Staubli VAL3: ALGORITH.pjx

--- ALGORITH.pjx ---
Parameters version=s7.3.1 stackSize=5000 millimeterUnit=true
Program file=ArcLength.pgx
Program file=Axis1Offset.pgx
Program file=ChangeCirPoint.pgx
Program file=ChangeCpoint.pgx
Program file=ChangeLength.pgx
Program file=CirClePoint.pgx
Program file=Circumcircle.pgx
Program file=Cshape.pgx
Program file=CutIn.pgx
Program file=CutOut.pgx
Program file=EllipsePoint.pgx
Program file=Facula.pgx
Program file=GetArcAngle.pgx
Program file=GetArcLength.pgx
Program file=GetClockwise.pgx
Program file=GetCutLength.pgx
Program file=GetWeldId.pgx
Program file=GetWeldReturn.pgx
Program file=HexagonPoint.pgx
Program file=Inscribedcircle.pgx
Program file=LineSym.pgx
Program file=LineSymArray.pgx
Program file=NoCloseShape.pgx
Program file=PentaclePoint.pgx
Program file=PentagonPoint.pgx
Program file=ReadMe.pgx
Program file=RectanglePoint.pgx
Program file=RegulPoint.pgx
Program file=SetFrame.pgx
Program file=start.pgx
Program file=stop.pgx
Program file=TrianglePoint.pgx
Program file=TubePoint.pgx
Data file=Algorith.dtx

--- ALGORITH.dtx ---
trsf trCut[100]
num nThickRadio = 100

--- start.pgx ---
program start()
  local trsf l_trTrsf[3]
  local trsf l_trTrsf1
  local num l_nNum
  local bool l_bBool
begin
  l_trTrsf[0]={0,1,0,0,0,0}
   l_trTrsf[1]={0,0,1,0,0,0}
   l_trTrsf[2]={1,0,0,0,0,0}



  call Circumcircle(l_trTrsf,l_trTrsf1,l_nNum,l_bBool)
  if !l_bBool
    popUpMsg("")
  else
    popUpMsg(toString(".5",l_nNum))
  endIf




end

--- ArcLength.pgx ---
public program ArcLength(trsf x_trFirst, trsf x_trCenter, trsf x_trEnd, num& x_nLength)
  local trsf l_trTrsf[3]
  local bool l_bBool
begin


  //获得圆弧长度
  //如果报错,那么就返回值为0


  x_nLength=0

  l_trTrsf[0]=x_trFirst
  l_trTrsf[1]=x_trCenter
  l_trTrsf[2]=x_trEnd

  call GetArcLength(l_trTrsf,x_nLength,l_bBool)
  if !l_bBool
    x_nLength=0
  endIf



end

--- Axis1Offset.pgx ---
public program Axis1Offset(pointRx& x_pP[], num x_nOffset, tool x_tTool)
  local num l_nNum
  local bool l_bMC
  local num l_nValue[3]
  local joint l_jJ
  local point l_pPoint
  local frame l_fFrame
begin
  if size(x_pP)<3
    return
  endIf

  for l_nNum=10 to size(x_pP)-3
    l_nValue[0]=(x_pP[l_nNum].trsf.x-x_pP[l_nNum+1].trsf.x)/(x_pP[l_nNum].trsf.x-x_pP[l_nNum+2].trsf.x)
    l_nValue[1]=(x_pP[l_nNum].trsf.y-x_pP[l_nNum+1].trsf.y)/(x_pP[l_nNum].trsf.y-x_pP[l_nNum+2].trsf.y)
    l_nValue[2]=(x_pP[l_nNum].trsf.z-x_pP[l_nNum+1].trsf.z)/(x_pP[l_nNum].trsf.z-x_pP[l_nNum+2].trsf.z)

    if l_nValue[0]!=l_nValue[1] or l_nValue[0]!=l_nValue[2]

      if !pointToJoint(x_tTool,herej(),x_pP[l_nNum],l_jJ)
        popUpMsg("转换出错")
        disablePower()
        return
      else
        l_jJ.j1=l_jJ.j1+x_nOffset
        link(l_fFrame,world)
        link(l_pPoint,world)
        l_pPoint.trsf=position(x_pP[l_nNum],world)

        l_fFrame.trsf=l_pPoint.trsf*!x_pP[l_nNum].trsf
        l_pPoint=jointToPoint(x_tTool,l_fFrame,l_jJ)
        x_pP[l_nNum].trsf=l_pPoint.trsf
      endIf




    endIf




  endFor

















end

--- ChangeCirPoint.pgx ---
public program ChangeCirPoint(trsf x_trCenter, num x_nDia, trsf& x_trSource, trsf x_trSupport, bool& x_bRes)
  local frame l_fFrame
  local point l_pPoint[3]
begin
  //根据边长和圆心点来修改相应的点。

  x_bRes=false

  if x_nDia<=0
    return
  endIf

  l_pPoint[0].trsf=x_trCenter
  l_pPoint[1].trsf=x_trSource
  l_pPoint[2].trsf=x_trSupport

  link(l_pPoint[0],world)
  link(l_pPoint[1],world)
  link(l_pPoint[2],world)
  link(l_fFrame,world)

  if setFrame(l_pPoint[0],l_pPoint[1],l_pPoint[2],l_fFrame)!=0
    return
  endIf

  l_pPoint[1].trsf=position(l_pPoint[1],l_fFrame)
  l_pPoint[1].trsf.x=x_nDia/2
  link(l_pPoint[1],l_fFrame)
  x_trSource=position(l_pPoint[1],world)
  x_bRes=true

end

--- ChangeCpoint.pgx ---
public program ChangeCpoint(trsf& x_trSource[], num x_nDia, bool& x_bRes)
  local trsf l_trTrsf
  local num l_nDia
  local num l_nNum
begin
  //根据直径来修改点的数值
  //外接圆

  //先根据三点来获得圆心点，然后根据三个点来求的圆心与三个点的长度。



  x_bRes=false

  if size(x_trSource)!=3
    return
  endIf


  call Circumcircle(x_trSource,l_trTrsf,l_nDia,x_bRes)
  if !x_bRes
    return
  endIf

  for l_nNum=0 to 2
    call ChangeCirPoint(l_trTrsf,x_nDia,x_trSource[l_nNum],x_trSource[sel(l_nNum==2,0,l_nNum+1)],x_bRes)
    if !x_bRes
      return
    endIf
  endFor

end

--- ChangeLength.pgx ---
public program ChangeLength(pointRx& x_trSource[], num& x_nLength[])
  local num l_nBuff[2]
begin


  //参数合法化处理
  if size(x_trSource)<3
    return
  endIf

  l_nBuff[0]=distance(x_trSource[0].trsf,x_trSource[1].trsf)
  l_nBuff[1]=distance(x_trSource[2].trsf,x_trSource[1].trsf)


  if x_nLength[1]<=0 or x_nLength[0]<=0 or l_nBuff[0]<=0 or l_nBuff[1]<=0
    return
  endIf



  x_trSource[0].trsf.x=(x_trSource[0].trsf.x-x_trSource[1].trsf.x)/l_nBuff[0]*x_nLength[0]+x_trSource[1].trsf.x
  x_trSource[0].trsf.y=(x_trSource[0].trsf.y-x_trSource[1].trsf.y)/l_nBuff[0]*x_nLength[0]+x_trSource[1].trsf.y
  x_trSource[0].trsf.z=(x_trSource[0].trsf.z-x_trSource[1].trsf.z)/l_nBuff[0]*x_nLength[0]+x_trSource[1].trsf.z

  x_trSource[2].trsf.x=(x_trSource[2].trsf.x-x_trSource[1].trsf.x)/l_nBuff[1]*x_nLength[1]+x_trSource[1].trsf.x
  x_trSource[2].trsf.y=(x_trSource[2].trsf.y-x_trSource[1].trsf.y)/l_nBuff[1]*x_nLength[1]+x_trSource[1].trsf.y
  x_trSource[2].trsf.z=(x_trSource[2].trsf.z-x_trSource[1].trsf.z)/l_nBuff[1]*x_nLength[1]+x_trSource[1].trsf.z









end

--- CirClePoint.pgx ---
public program CirClePoint(trsf x_trCenter, num x_nDia, trsf& x_trDest[], bool& x_bRes)
  local num l_nNum
  local frame l_fFrame
  local point l_pP
begin
  //由圆心直径获得圆的四个点
  //是通过逆时针来获得

  x_bRes=false

  if x_nDia<=0
    return
  endIf

  link(l_fFrame,world)
  l_fFrame.trsf=x_trCenter
  link(l_pP,l_fFrame)


  //第一个点
  l_pP.trsf={0,0,0,0,0,0}
  l_pP.trsf.y=-x_nDia/2
  x_trDest[0]=position(l_pP,world)


  //第二个点
  l_pP.trsf={0,0,0,0,0,0}
  l_pP.trsf.x=x_nDia/2
  x_trDest[1]=position(l_pP,world)



  //第三个点
  l_pP.trsf={0,0,0,0,0,0}
  l_pP.trsf.y=x_nDia/2
  x_trDest[2]=position(l_pP,world)


  //第四个点
  l_pP.trsf={0,0,0,0,0,0}
  l_pP.trsf.x=-x_nDia/2
  x_trDest[3]=position(l_pP,world)

   x_trDest[4]= x_trDest[0]





  //圆心点
  x_trDest[20]=x_trCenter

  x_bRes=true

  //辅助点
  l_pP.trsf={0,0,0,0,0,0}
  l_pP.trsf.y=-x_nDia/2
    l_pP.trsf.x=x_nDia/2
  x_trDest[9]=position(l_pP,world)






end

--- Circumcircle.pgx ---
public program Circumcircle(trsf& x_trSource[], trsf& x_trCenter, num& x_nDia, bool& x_bRes)
  local point l_pPoint[3]
  local num l_ni
  local frame l_fFrame
  local point l_pCenter
  local num x1
  local num x2
  local num x3
  local num y1
  local num y2
  local num y3
begin
  //由圆的三点获得圆的圆心与直径
  //外接圆圆心

 call SetFrame(x_trSource,l_fFrame,x_bRes)
 if !x_bRes
  return
endIf

  //外接圆圆心与直径


  //参数传递
  for l_ni=0 to 2
    l_pPoint[l_ni].trsf=x_trSource[l_ni]
    link(l_pPoint[l_ni],world)
    l_pPoint[l_ni].trsf=position(l_pPoint[l_ni],l_fFrame)
  endFor



  //如果原点的坐标不是三个零，则报错
  if l_pPoint[0].trsf.x!=0 or l_pPoint[0].trsf.y!=0 or  l_pPoint[0].trsf.z!=0
    x_bRes=false
    return
  endIf


//利用公式求圆心

//******************************************
//求圆公式
  x1=l_pPoint[0].trsf.x
  x2=l_pPoint[1].trsf.x
  x3=l_pPoint[2].trsf.x
  y1=l_pPoint[0].trsf.y
  y2=l_pPoint[1].trsf.y
  y3=l_pPoint[2].trsf.y


  if((x3-x1)*(y2-y1)-(x2-x1)*(y3-y1))!=0
    link(l_pCenter,l_fFrame)
    l_pCenter.trsf={0,0,0,0,0,0}
    l_pCenter.trsf.x=((y2-y1)*(y3*y3-y1*y1+x3*x3-x1*x1)-(y3-y1)*(y2*y2-y1*y1+x2*x2-x1*x1))/(2*(x3-x1)*(y2-y1)-2*(x2-x1)*(y3-y1))
    l_pCenter.trsf.y=((x2-x1)*(x3*x3-x1*x1+y3*y3-y1*y1)-(x3-x1)*(x2*x2-x1*x1+y2*y2-y1*y1))/(2*(y3-y1)*(x2-x1)-2*(y2-y1)*(x3-x1))
    x_trCenter=position(l_pCenter,world)
    x_nDia=2*distance(l_pCenter.trsf,l_pPoint[0].trsf)
    x_bRes=x_nDia>0
  else
    x_bRes=false
    return
  endIf
//**********************************************

end

--- CSHAPE.pgx ---
public program Cshape(trsf& x_Source[], trsf& x_trCut[], num x_nAngle, num& x_nPointCout, trsf x_trCen, num x_nDia, bool& x_bRes)
  local trsf l_trTrsf[3]
  local num l_nNum
  local num l_nBuff
  local trsf l_trBuff
  local frame l_fFrame
begin

  //C型图形
  x_bRes=false
  if x_nAngle<=0 or x_nAngle>3600

    return
  endIf

  //由于TRSF.RZ的范围是 +-360


  l_trTrsf[0]=x_trCen
  l_trTrsf[1]=x_Source[0]
  l_trTrsf[2]=x_Source[1]

  // x_trCut[0]=x_Source[0]
  call SetFrame(l_trTrsf,l_fFrame,x_bRes)
  if !x_bRes
    return
  endIf


  x_nPointCout=roundUp(x_nAngle/180)+1
  x_nDia=x_nDia/2
  l_nBuff=x_nAngle/(x_nPointCout-1)/2
//  nNum=l_nBuff
  x_trCut[0]=l_fFrame.trsf*{x_nDia,0,0,0,0,0}
  for l_nNum=0 to x_nPointCout-2
    x_trCut[l_nNum*2+1]=l_fFrame.trsf*{cos((l_nNum*2+1)*l_nBuff)*x_nDia,sin((l_nNum*2+1)*l_nBuff)*x_nDia,0,0,0,0}
    x_trCut[l_nNum*2+2]=l_fFrame.trsf*{cos((l_nNum*2+2)*l_nBuff)*x_nDia,sin((l_nNum*2+2)*l_nBuff)*x_nDia,0,0,0,0}

  endFor


  x_bRes=true




end

--- CUTIN.pgx ---
public program CutIn(trsf x_trCenter, trsf& x_trLine[], trsf& x_trDest[], trsf& x_trCut, num x_nType, num x_nPercent, bool& x_bRes)
  local pointRx l_trCutInP
  local frame l_fFrame
  local trsf l_trBuff[3]
  local num l_nR
begin
  //切入引线
  //x_nType==0  无引线
  //==1   直线
  //==2   圆弧


  //如果是直线，直接退出
  if x_nType==0
    x_bRes=true
    return
  else
    x_bRes=false
  endIf


  //参数合法性判断
  if x_nType<0 or x_nType>2
    return
  endIf



  //根据三点求用户坐标系
  l_trBuff[0]=x_trLine[0]
  l_trBuff[1]=x_trLine[1]
  l_trBuff[2]=x_trCenter

  call SetFrame(l_trBuff,l_fFrame,x_bRes)
  if !x_bRes
    return
  endIf

  //**********************************
  //2014.10.23
  //从圆心开始调整
  //为切厚板改写的程序
  if  x_nPercent==101
    //2015.01.22
    //添加新的变量来支持厚板切割
    //厚板切割内切圆的圆心的长度
    if distance(x_trLine[0],x_trCenter)<=max(5,nThickRadio)
      x_trDest[0]=x_trCenter
    else
      l_trCutInP.trsf={0,10,0,0,0,0}
      link(l_trCutInP,l_fFrame)
      x_trDest[0]=position(l_trCutInP,world)
    endIf
    return
  endIf

  //*********************************





  l_trCutInP.trsf=x_trCenter
  link(l_trCutInP,world)
  l_trCutInP.trsf=position(l_trCutInP,l_fFrame)
  //2014.7.24
  l_nR=min(abs(l_trCutInP.trsf.y)/2,10)
  //l_nR=min(abs(l_trCutInP.trsf.y),10)


  if l_nR==0
    x_bRes=false
    return
  endIf

  //切入切出比例
  if x_nPercent>0 and x_nPercent<100

    l_nR=l_nR*x_nPercent/100
  endIf


  l_trCutInP.trsf.y=0
  link(l_trCutInP,l_fFrame)
  l_trCutInP.trsf=position(l_trCutInP,world)

  x_trCut=l_trCutInP.trsf


  l_trBuff[0]=l_trCutInP.trsf
  call SetFrame(l_trBuff,l_fFrame,x_bRes)
  if !x_bRes
    return
  endIf

  l_trCutInP.trsf={-l_nR,l_nR,0,0,0,0}
  link(l_trCutInP,l_fFrame)
  x_trDest[0]=position(l_trCutInP,world)

  if x_nType==2
    l_trCutInP.trsf={-sin(45)*l_nR,l_nR-sin(45)*l_nR,0,0,0,0}
    link(l_trCutInP,l_fFrame)
    x_trDest[1]=position(l_trCutInP,world)
  endIf

end

--- CUTOUT.pgx ---
public program CutOut(trsf x_trCenter, trsf& x_trLine[], trsf& x_trDest[], trsf& x_trCut, num x_nType, num x_nPercent, bool& x_bRes)
  local trsf l_trTrsf[2]
begin
  //切入引线
    if x_nType==0
    x_bRes=true
    return
    endIf
  call CutIn(x_trCenter,x_trLine,l_trTrsf,x_trCut,x_nType,x_nPercent,x_bRes)
  if !x_bRes
    return
  endIf

  x_trLine[1]=x_trLine[0]
  x_trLine[0]=x_trCenter


  call LineSymArray(l_trTrsf,x_trLine,x_trDest,x_bRes)


end

--- EllipsePoint.pgx ---
public program EllipsePoint(trsf& x_trSource[], trsf& x_trDest[], bool& x_bRes)
  local frame l_fFrame
  local num l_Dia
  local num l_nLegth
  local point l_pBuff
begin
  //腰形孔

  //根据三个trsf建立frame
  call SetFrame(x_trSource,l_fFrame,x_bRes)
  if !x_bRes
    return
  endIf
 link(l_fFrame,world)

  //圆弧的直径
  l_Dia=distance(x_trSource[1],x_trSource[2])
  l_nLegth=distance(x_trSource[0],x_trSource[1])



  link(l_pBuff,l_fFrame)
  l_pBuff.trsf={l_nLegth/2,0,0,0,0,0}
  x_trDest[0]=position(l_pBuff,world)

  l_pBuff.trsf={l_nLegth,0,0,0,0,0}
  x_trDest[1]=position(l_pBuff,world)

  l_pBuff.trsf={l_nLegth+l_Dia/2,l_Dia/2,0,0,0,0}
  x_trDest[2]=position(l_pBuff,world)

  l_pBuff.trsf={l_nLegth,l_Dia,0,0,0,0}
  x_trDest[3]=position(l_pBuff,world)

  l_pBuff.trsf={0,l_Dia,0,0,0,0}
  x_trDest[4]=position(l_pBuff,world)

  l_pBuff.trsf={-l_Dia/2,l_Dia/2,0,0,0,0}
  x_trDest[5]=position(l_pBuff,world)

  l_pBuff.trsf={0,0,0,0,0,0}
  x_trDest[6]=position(l_pBuff,world)

  x_trDest[7]=x_trDest[0]


    //圆心点
  l_pBuff.trsf={l_nLegth/2,min(l_nLegth/2,l_Dia/2),0,0,0,0}
  x_trDest[20]=position(l_pBuff,world)



  x_bRes=true

end

--- FACULA.pgx ---
public program Facula(trsf& x_trSource[], num x_nDia, num x_nType, trsf& x_trDownLead, bool& x_bRes)
  local trsf l_trTrsf
  local num l_nDia
  local num l_nNum
begin
  //光斑补偿

  if  x_nDia<=0 or x_nType==10 or x_nType==9
     x_bRes=true
     return
  endIf

  //光斑强制设置为0.1
  if x_nDia>1
    x_nDia=0.1
  endIf


  if x_nType==2
    x_trDownLead.ry=max(x_trDownLead.ry-x_nDia,0.1)
    x_bRes=true
    return
  endIf

  if x_nType==12
    x_trDownLead.ry=x_trDownLead.ry+x_nDia
    x_bRes=true
    return
  endIf

  l_nDia=0

  call Circumcircle(x_trSource,l_trTrsf,l_nDia,x_bRes)
  if !x_bRes
    return
  endIf

  if x_nDia>=l_nDia/2
    x_nDia=0
    x_bRes=true
    return
  endIf


  switch x_nType
    case 1,3,4,5,6,7,8

      l_nDia=l_nDia-x_nDia*2
    break

    case 11,13,14,15,16,17,18
      l_nDia=l_nDia+x_nDia*2

    break

  endSwitch


  call ChangeCpoint(x_trSource,l_nDia,x_bRes)

end

--- GetArcAngle.pgx ---
public program GetArcAngle(trsf x_trTCent, trsf x_trX, trsf x_trY, num& x_nAngle, bool& x_bRes)
  local num l_nDia
  local num l_nLength
  local trsf l_trCenter
  local trsf l_trSource[3]
begin

  l_trSource[0]=x_trTCent
  l_trSource[1]=x_trX
  l_trSource[2]=x_trY


    call Circumcircle(l_trSource,l_trCenter,l_nDia,x_bRes)
  if !x_bRes or l_nDia<=0
    x_bRes=false
    return
  endIf

  l_nLength=distance(l_trSource[0],l_trSource[2])

  if l_nLength>=l_nDia

    x_nAngle=180
  else
      x_nAngle=asin(l_nLength/l_nDia)
  endIf





end

--- GetArcLength.pgx ---
public program GetArcLength(trsf& x_trSource[], num& x_nLength, bool& x_bRes)
  local frame l_fFrame
  local trsf l_trCenter
  local num l_nDia
  local num l_nLength
  local num l_nAngle
  local trsf l_trBuff
begin
  //获得圆弧长度

  call Circumcircle(x_trSource,l_trCenter,l_nDia,x_bRes)
  if !x_bRes or l_nDia<=0
    x_bRes=false
    return
  endIf






  //计算三点的圆弧长度
  //2015.09.09
  //

  //强制二分，避免出现多边弧的问题
  l_trBuff=interpolateC(x_trSource[0],x_trSource[1],x_trSource[2],0.5)



  l_nLength=distance(x_trSource[0],l_trBuff)
  l_nAngle=asin(l_nLength/l_nDia)
  x_nLength=l_nAngle/180*l_nLength


  l_nLength=distance(l_trBuff,x_trSource[2])
  l_nAngle=asin(l_nLength/l_nDia)
  x_nLength=l_nAngle/180*l_nLength+x_nLength








end

--- GetClockwise.pgx ---
public program GetClockwise(trsf& x_trSource[], trsf& x_trRes, bool& x_bRes)
  local frame l_fFrame
  local trsf l_trBuff[3]
  local num l_nNum
  local pointRx l_pP
begin
  //获得三个点是否是顺时针还是逆时针
  //获得顺时针与逆时针的方向
  //主要是RX,RY,RZ

  //  设   p1=(x1,y1)，   p2=(x2,y2)，   p3=(x3,y3)
  //
  //  求向量
  //          p12=(x2-x1,y2-y1)
  //          p23=(x3-x2,y3-y2)
  //
  //  则当   p12   与   p23   的叉乘（向量积）
  //
  //      p12   x   p23   =   (x2-x1)*(y3-y2)-(y2-y1)*(x3-x2)
  //
  //  为正时，p1-p2-p3   路径的走向为逆时针，
  //  为负时，p1-p2-p3   走向为顺时针，
  //  为零时，p1-p2-p3   所走的方向不变，亦即三点在一直线上。



  for l_nNum=0 to 2
    l_trBuff[l_nNum]=x_trSource[l_nNum]
  endFor

  //  //(x2-x1)*(y3-y2)-(y2-y1)*(x3-x2)
  //  if((l_trBuff[1].x-l_trBuff[0].x)*(l_trBuff[2].y-l_trBuff[1].y)-(l_trBuff[2].x-l_trBuff[1].x)*(l_trBuff[1].y-l_trBuff[0].y))>0
  //    //如果路径的走向为逆时针，
  //    for l_nNum=0 to 2
  //      l_trBuff[l_nNum]=x_trSource[2-l_nNum]
  //    endFor
  //  endIf
  call SetFrame(l_trBuff,l_fFrame,x_bRes)
  if !x_bRes
    return
  endIf

  if abs($rotAngle(!l_trBuff[0]*l_fFrame.trsf))<90

    x_trRes=l_fFrame.trsf
    x_bRes=true
    return

  endIf

  for l_nNum=0 to 2
    l_trBuff[l_nNum]=x_trSource[2-l_nNum]
  endFor

  call SetFrame(l_trBuff,l_fFrame,x_bRes)
  if !x_bRes
    return
  endIf
  x_trRes=l_fFrame.trsf
  x_bRes=true


  //  l_trBuff[0]={0,0,0,l_trBuff[0].rx,l_trBuff[0].ry,0}
  //  l_trBuff[1]={0,0,0,l_fFrame.trsf.rx,l_fFrame.trsf.ry,0}
  //  l_nNum=$rotAngle(!l_trBuff[0]*l_trBuff[1])
  //  if abs(l_nNum)<90
  //    x_trRes=l_fFrame.trsf
  //  else
  //
  //    //判断
  //        for l_nNum=0 to 2
  //      l_trBuff[l_nNum]=x_trSource[2-l_nNum]
  //    endFor
  //
  //  call SetFrame(l_trBuff,l_fFrame,x_bRes)
  //  if !x_bRes
  //    return
  //  endIf
  //  l_trBuff[0]={0,0,0,l_trBuff[0].rx,l_trBuff[0].ry,0}
  //  l_trBuff[1]={0,0,0,l_fFrame.trsf.rx,l_fFrame.trsf.ry,0}
  //  l_nNum=$rotAngle(!l_trBuff[0]*l_trBuff[1])
  //    if abs(l_nNum)>90
  //      x_bRes=false
  //      return
  //
  //    endIf
  //    x_trRes=l_fFrame.trsf
  //    x_bRes=true
  //
  //  endIf

end

--- GetCutLength.pgx ---
public program GetCutLength(point& x_pCut[], point& x_pMC[], bool& x_bMC[], num& x_nLength, bool& x_bRes)
  local num l_nNum
  local trsf l_trBuff[3]
  local trsf l_trTe
  local num l_nArc
begin
  //获得切割的真正长度是多少



  x_bRes=false
  x_nLength=0
  if size(x_pCut)!=size(x_pMC) or size(x_pCut)!=size(x_bMC)
    return
  endIf

  //如果只有一个点，则退出
   if size(x_bMC)==1
    x_bRes=true
    return
  endIf


  //多于一个点进行计算
  for l_nNum=1 to size(x_bMC)-1


    if !x_bMC[l_nNum]
      x_nLength=distance(x_pCut[l_nNum-1].trsf,x_pCut[l_nNum].trsf)+x_nLength

    else
      l_trBuff[0]=x_pCut[l_nNum-1].trsf
      l_trBuff[1]=x_pMC[l_nNum].trsf
      l_trBuff[2]=x_pCut[l_nNum].trsf
      //获取圆弧长度
      call GetArcLength(l_trBuff,l_nArc,x_bRes)
      if !x_bRes
        return
      endIf
      x_nLength=x_nLength+l_nArc

    endIf


  endFor

  x_bRes=true

end

--- GetWeldId.pgx ---
public program GetWeldId(point& x_pCut[], point& x_pMC[], bool& x_bMC[], num x_nLength, num& x_nMoveId, bool& x_bRes, num x_nWeldEndOffse)
  local num l_nNum
  local num l_nBuffLength
  local trsf l_trBuff[3]
  local num l_nArc
  local num l_nBuff
begin
  //焊接的收弧点的moveid

  //x_nLength   收弧长度
  //关键函数



  x_nMoveId=0
  x_bRes=false

  if size(x_pCut)<2 or size(x_bMC)!=size(x_pCut) or size(x_bMC)!=size(x_pCut)
    return
  endIf


  if x_nLength<=0
    //    x_nMoveId=0
    ////    x_bRes=true
    //    return
    x_nLength=5
  endIf





  //实际走的长度
  //2014.04.10
  // 可以对长度经修正




  //x_nWeldEndOffse=min(max(0.1,x_nWeldEndOffse),40)
  ////2015.09.08
  ////强制设置为o
  //x_nWeldEndOffse=0


  //if size(x_bMC)>1
  //  if distance(x_pCut[size(x_pCut)-1].trsf,x_pCut[size(x_pCut)-2].trsf)<30
  //    x_nWeldEndOffse=0
  //  endIf
  //else
  //  x_nMoveId=1
  //  x_bRes=true
  //  return
  //endIf

  //  x_nLength=max(0.1,l_nNum-x_nLength-x_nWeldEndOffse)

  //************************


  //反算，从结尾开始算
  l_nBuffLength=0
  for l_nNum=size(x_bMC)-1 to 1 step -1
    if !x_bMC[l_nNum]
      l_nArc=distance(x_pCut[l_nNum-1].trsf,x_pCut[l_nNum].trsf)
      l_nBuffLength=l_nArc+l_nBuffLength
    else
      l_trBuff[0]=x_pCut[l_nNum-1].trsf
      l_trBuff[1]=x_pMC[l_nNum].trsf
      l_trBuff[2]=x_pCut[l_nNum].trsf
      call GetArcLength(l_trBuff,l_nArc,x_bRes)
      if !x_bRes
        return
      endIf
      l_nBuffLength=l_nBuffLength+l_nArc
    endIf

    if l_nBuffLength>=x_nLength

      //这句是重点
      //容易计算错误
      x_nMoveId=l_nNum+(l_nBuffLength-x_nLength)/l_nArc
      x_bRes=true
      return
    endIf
  endFor

  //跳出整个程序
  return







  //顺算，从头开始算
  //获取整个长度
  call GetCutLength(x_pCut,x_pMC,x_bMC,l_nNum,x_bRes)
  if !x_bRes or l_nNum<=0 or x_nLength>=l_nNum
    return
  endIf

  x_nLength=l_nNum-x_nLength
  l_nBuffLength=0
  for l_nNum=1 to size(x_bMC)-1
    if !x_bMC[l_nNum]
      l_nArc=distance(x_pCut[l_nNum-1].trsf,x_pCut[l_nNum].trsf)
      l_nBuffLength=l_nArc+l_nBuffLength
    else
      l_trBuff[0]=x_pCut[l_nNum-1].trsf
      l_trBuff[1]=x_pMC[l_nNum].trsf
      l_trBuff[2]=x_pCut[l_nNum].trsf
      call GetArcLength(l_trBuff,l_nArc,x_bRes)
      if !x_bRes
        return
      endIf
      l_nBuffLength=l_nBuffLength+l_nArc
    endIf


    if l_nBuffLength>x_nLength
      x_nMoveId=l_nNum-((l_nBuffLength-x_nLength)/l_nArc)+1
      // x_nMoveId=l_nNum+()
      x_bRes=true
      return
    endIf

    l_nBuff=l_nBuffLength

  endFor








  x_bRes=false

end

--- GetWeldReturn.pgx ---
public program GetWeldReturn(point& x_pCut[], point& x_pMC[], bool& x_bMC[], num x_nId, num& x_nReturnId, num x_nLength, bool& x_bRes)
  local num l_nNum
  local trsf l_trBuff[3]
  local trsf l_trTe
  local num l_nArc
  local num l_nLength
  local num l_nWeld
begin
  //获得回退点的MOVEID



  x_bRes=false
  x_nReturnId=-1
  if size(x_pCut)!=size(x_pMC) or size(x_pCut)!=size(x_bMC) or size(x_bMC)<(x_nId-1) or x_nLength<=0
    return
  endIf

  //如果只有一个点，则退出
   if size(x_bMC)==1
    x_bRes=true
    return
  endIf

  if roundDown(x_nId)==roundUp(x_nId)
      x_nId=x_nId+0.00001
  endIf


  //多于一个点进行计算
  l_nLength=0
  for l_nNum=1 to roundDown(x_nId)


    if !x_bMC[l_nNum]
      l_nArc=distance(x_pCut[l_nNum-1].trsf,x_pCut[l_nNum].trsf)

    else
      l_trBuff[0]=x_pCut[l_nNum-1].trsf
      l_trBuff[1]=x_pMC[l_nNum].trsf
      l_trBuff[2]=x_pCut[l_nNum].trsf
      //获取圆弧长度
      call GetArcLength(l_trBuff,l_nArc,x_bRes)
      if !x_bRes
        return
      endIf
    endIf

    //取余
    if l_nNum==roundDown(x_nId)
      l_nLength=(x_nId-l_nNum)*l_nArc+l_nLength
    else
      l_nLength=l_nLength+l_nArc
    endIf
  endFor

 // popUpMsg(toString(".3",l_nLength))
  //需要达到点的号码
  if l_nLength<=x_nLength
    x_nReturnId=1
      x_bRes=true
    return
  else
    l_nWeld=l_nLength-x_nLength
  endIf



  l_nLength=0
  for l_nNum=1 to roundUp(x_nId)


    if !x_bMC[l_nNum]
      l_nArc=distance(x_pCut[l_nNum-1].trsf,x_pCut[l_nNum].trsf)

    else
      l_trBuff[0]=x_pCut[l_nNum-1].trsf
      l_trBuff[1]=x_pMC[l_nNum].trsf
      l_trBuff[2]=x_pCut[l_nNum].trsf
      //获取圆弧长度
      call GetArcLength(l_trBuff,l_nArc,x_bRes)
      if !x_bRes
        return
      endIf
    endIf



    if l_nNum==roundUp(x_nId)-1
      l_nLength=(x_nId-roundDown(x_nId))*l_nArc+l_nLength
    else
      l_nLength=l_nLength+l_nArc
    endIf

    if l_nLength>=l_nWeld
      x_nReturnId=l_nNum-1-(l_nLength-l_nWeld)/l_nArc

        x_bRes=true
      return
    endIf
  endFor

  x_bRes=false

end

--- HexagonPoint.pgx ---
public program HexagonPoint(trsf& x_trSource[], trsf& x_trDest[], bool& x_bRes)
  local frame l_fFrame
  local num l_Dia
  local num l_nLegth
  local point l_pBuff
begin
  //六边形

  //根据三个trsf建立frame

  call SetFrame(x_trSource,l_fFrame,x_bRes)
  if !x_bRes
    return
  endIf


  //圆弧的直径
  l_Dia=distance(x_trSource[1],x_trSource[2])
  l_nLegth=distance(x_trSource[0],x_trSource[1])


  //算出点
  link(l_pBuff,l_fFrame)
  l_pBuff.trsf={l_nLegth/2,0,0,0,0,0}
  x_trDest[0]=position(l_pBuff,world)

  l_pBuff.trsf={l_nLegth,0,0,0,0,0}
  x_trDest[1]=position(l_pBuff,world)

//  l_pBuff.trsf={l_nLegth+sin(15)*l_nLegth,cos(15)*l_nLegth,0,0,0,0}
//  x_trDest[2]=position(l_pBuff,world)
//
//  l_pBuff.trsf={l_nLegth,2*cos(15)*l_nLegth,0,0,0,0}
//  x_trDest[3]=position(l_pBuff,world)
//
//  l_pBuff.trsf={0,2*cos(15)*l_nLegth,0,0,0,0}
//  x_trDest[4]=position(l_pBuff,world)
//
//  l_pBuff.trsf={-sin(15)*l_nLegth,sin(75)*l_nLegth,0,0,0,0}
//  x_trDest[5]=position(l_pBuff,world)

  //2013.10.15  修改了正六边形算法
    l_pBuff.trsf={l_nLegth+sin(30)*l_nLegth,cos(30)*l_nLegth,0,0,0,0}
  x_trDest[2]=position(l_pBuff,world)

  l_pBuff.trsf={l_nLegth,2*cos(30)*l_nLegth,0,0,0,0}
  x_trDest[3]=position(l_pBuff,world)

  l_pBuff.trsf={0,2*cos(30)*l_nLegth,0,0,0,0}
  x_trDest[4]=position(l_pBuff,world)

  l_pBuff.trsf={-sin(30)*l_nLegth,sin(60)*l_nLegth,0,0,0,0}
  x_trDest[5]=position(l_pBuff,world)



  l_pBuff.trsf={0,0,0,0,0,0}
  x_trDest[6]=position(l_pBuff,world)

  x_trDest[7]=x_trDest[0]


  //圆心点
  l_pBuff.trsf={l_nLegth/2,l_nLegth/2/sin(30),0,0,0,0}
  x_trDest[20]=position(l_pBuff,world)

  x_bRes=true

end

--- Inscribedcircle.pgx ---
public program Inscribedcircle(trsf& x_trSource[], trsf& x_trCenter, num& x_nDia, bool& x_bRes)
  local num l_ni
  local frame l_fFrame
  local point l_pCenter
  local num a
  local num b
  local num c
  local num p
  local num s
  local num r
  local num l_angle
begin
  //由三角形求内切圆圆心
  //内切圆圆心
  x_bRes=false
  a=distance(x_trSource[0],x_trSource[1])
  b=distance(x_trSource[1],x_trSource[2])
  c=distance(x_trSource[0],x_trSource[2])
  p=(a+b+c)/2
  s=sqrt(p*(p-a)*(p-b)*(p-c))
  r=s/p
  l_angle=acos((c*c+a*a-b*b)/2/a/c)/2

  if l_angle<0
    return
  endIf


  call SetFrame(x_trSource,l_fFrame,x_bRes)
  if !x_bRes
    return
  endIf

  link(l_pCenter,l_fFrame)
  l_pCenter.trsf={r/tan(l_angle),r,0,0,0,0}
  x_trCenter=position(l_pCenter,world)
  x_nDia=r
end

--- LINESYM.pgx ---
public program LineSym(trsf x_trSource, trsf& x_trLine[], trsf& x_trDest, bool& x_bRes)
  local frame l_fFrame
  local point l_p
  local trsf l_trT[3]
begin

  //有关直线对称


  l_trT[0]=x_trLine[0]
  l_trT[1]=x_trLine[1]
  l_trT[2]=x_trSource

  call SetFrame(l_trT,l_fFrame,x_bRes)
  if !x_bRes
    return
  endIf

  l_p.trsf=x_trSource
  link(l_p,world)
  l_p.trsf=position(l_p,l_fFrame)
  l_p.trsf.y=-l_p.trsf.y
  link(l_p,l_fFrame)
  x_trDest=position(l_p,world)



end

--- LineSymArray.pgx ---
public program LineSymArray(trsf& x_trSource[], trsf& x_trLine[], trsf& x_trDest[], bool& x_bRes)
  local num l_nNum
begin

  //点的数组有关直线对称
  for l_nNum=0 to size(x_trSource)-1
    call LineSym(x_trSource[l_nNum],x_trLine,x_trDest[l_nNum],x_bRes)
    if !x_bRes
      return
    endIf
  endFor
end

--- NoCloseShape.pgx ---
public program NoCloseShape(point& x_pCut[], point& x_pMC[], bool& x_bMC[], num x_nLength, bool& x_bRes)
  local num l_nNum
  local trsf l_trBuff[3]
  local trsf l_trTe
  local num l_nArc
  local num l_nLength
begin
  //获得切割的真正长度是多少



  x_bRes=false
  //  x_nLength=0
  if size(x_pCut)!=size(x_pMC) or size(x_pCut)!=size(x_bMC)
    return
  endIf

  //如果只有一个点，则退出
  if size(x_bMC)==1
    //  x_bRes=true
    return
  endIf


  //多于一个点进行计算
  l_nNum=size(x_bMC)-1
  if !x_bMC[l_nNum]
    l_nLength=distance(x_pCut[l_nNum-1].trsf,x_pCut[l_nNum].trsf)

  else
    l_trBuff[0]=x_pCut[l_nNum-1].trsf
    l_trBuff[1]=x_pMC[l_nNum].trsf
    l_trBuff[2]=x_pCut[l_nNum].trsf
    //获取圆弧长度
    call GetArcLength(l_trBuff,l_nLength,x_bRes)
    if !x_bRes
      return
    endIf

  endIf

  if x_nLength>l_nLength
    x_bRes=false
    return
  endIf

  if !x_bMC[l_nNum]
    l_trTe=interpolateL(x_pCut[l_nNum-1].trsf,x_pCut[l_nNum].trsf,x_nLength/l_nLength)
    x_pCut[l_nNum].trsf=l_trTe
  else

    l_trTe=interpolateC(x_pCut[l_nNum-1].trsf,x_pMC[l_nNum].trsf,x_pCut[l_nNum].trsf,x_nLength/l_nLength)
    //保证其是小于180度的圆弧
    if distance(l_trTe,x_pCut[l_nNum-1].trsf)<=distance(x_pMC[l_nNum].trsf,x_pCut[l_nNum-1].trsf)
      x_pCut[l_nNum].trsf=x_pMC[l_nNum].trsf
      x_pMC[l_nNum].trsf=l_trTe
    else
      x_pCut[l_nNum].trsf=l_trTe
    endIf



  endIf



  x_bRes=true

end

--- PentaclePoint.pgx ---
public program PentaclePoint(trsf& x_trSource[], trsf& x_trDest[], bool& x_bRes)
  local num l_ni
  local frame l_fFrame
  local num l_Dia
  local num l_nLegth
  local point l_pBuff
  local trsf l_trBuff[3]
  local num l_nNum
begin
  //五角星

  //根据三个trsf建立frame
  call SetFrame(x_trSource,l_fFrame,x_bRes)
  if !x_bRes
    return
  endIf


  //圆弧的直径
  l_nLegth=distance(x_trSource[0],x_trSource[1])

  link(l_pBuff,l_fFrame)
  l_pBuff.trsf={l_nLegth/2,tan(54)*l_nLegth/2,0,0,0,0}
  l_trBuff[0]=position(l_pBuff,world)

  l_pBuff.trsf={l_nLegth/2,tan(36)*l_nLegth/2,0,0,0,0}
  l_trBuff[1]=position(l_pBuff,world)

  l_pBuff.trsf={l_nLegth,0,0,0,0,0}
  l_trBuff[2]=position(l_pBuff,world)

  //根据求的三点建立新的frame
    call SetFrame(l_trBuff,l_fFrame,x_bRes)
  if !x_bRes
    return
  endIf
  l_Dia=distance(l_trBuff[0],l_trBuff[1])
  l_nLegth=distance(l_trBuff[0],l_trBuff[2])


    link(l_pBuff,l_fFrame)
   for l_ni=0 to 9
    l_nNum=sel(l_ni%2==0,l_Dia,l_nLegth)
    l_pBuff.trsf={l_nNum*cos(36*l_ni),sin(36*l_ni)*l_nNum,0,0,0,0}
    x_trDest[l_ni]=position(l_pBuff,world)
  endFor
   x_trDest[10]=x_trDest[0]



end

--- PentagonPoint.pgx ---
public program PentagonPoint(trsf& x_trSource[], trsf& x_trDest[], bool& x_bRes)
  local point l_pPoint[3]
  local num l_ni
  local frame l_fFrame
  local num l_Dia
  local num l_nLegth
  local point l_pBuff
begin
  //五边形
  //根据三个trsf建立frame
  call SetFrame(x_trSource,l_fFrame,x_bRes)
  if !x_bRes
    return
  endIf

  //圆弧的直径
//  l_Dia=distance(x_trSource[1],x_trSource[2])
  l_nLegth=distance(x_trSource[0],x_trSource[1])



  link(l_pBuff,l_fFrame)
  l_pBuff.trsf={l_nLegth/2,0,0,0,0,0}
  x_trDest[0]=position(l_pBuff,world)

  l_pBuff.trsf={l_nLegth,0,0,0,0,0}
  x_trDest[1]=position(l_pBuff,world)

//  l_pBuff.trsf={l_nLegth+sin(18)*l_nLegth,cos(18)*l_nLegth,0,0,0,0}
//  x_trDest[2]=position(l_pBuff,world)
//
//  l_pBuff.trsf={l_nLegth/2,(sin(36)+sin(54))*l_nLegth,0,0,0,0}
//  x_trDest[3]=position(l_pBuff,world)
//
//  l_pBuff.trsf={-sin(36)*l_nLegth,cos(36)*l_nLegth,0,0,0,0}
//  x_trDest[4]=position(l_pBuff,world)
//

//2013.10.26
  l_pBuff.trsf={l_nLegth+sin(18)*l_nLegth,cos(18)*l_nLegth,0,0,0,0}
  x_trDest[2]=position(l_pBuff,world)

  l_pBuff.trsf={l_nLegth/2,(sin(36)+sin(72))*l_nLegth,0,0,0,0}
  x_trDest[3]=position(l_pBuff,world)

  l_pBuff.trsf={-sin(18)*l_nLegth,cos(18)*l_nLegth,0,0,0,0}
  x_trDest[4]=position(l_pBuff,world)




//*************************************

  l_pBuff.trsf={0,0,0,0,0,0}
  x_trDest[5]=position(l_pBuff,world)

  x_trDest[6]=x_trDest[0]

    //圆心点
  l_pBuff.trsf={l_nLegth/2,l_nLegth/2/sin(36),0,0,0,0}
  x_trDest[20]=position(l_pBuff,world)



end

--- README.pgx ---
program ReadMe()
begin
  //利用trsf来实现图形变换的函数库
  //支持切圆管，三角形，圆，矩形，正五边形，正六边形，腰圆，五角星，切圆管
  //一般规则图形使用三个点来实现，除了圆心-直径法以外
  //直接客户根据三点法来实现自定义规则类型


  //TrianglePoint  三角形
  //SetFrame  通过三个点来建立frame
  //LineSym 点关于线对称
  //ChangeCirPoint   根据圆心，直径来修改点的位置
  //CirClePoint  根据圆心 直径来求的两个movec的点
  //Circumcircle 内切圆
  //Cshape  C型图形 主要是为焊接使用
  //CutIn   切入引线
  //CutOut   切出引线


  //TubePoint 切割圆管
  //TrianglePoint  三角形
  //RectanglePoint


//Val3进行图形算法库





end

--- RectanglePoint.pgx ---
public program RectanglePoint(trsf& x_trSource[], trsf& x_trDest[], bool& x_bRes)
  local frame l_fFrame
  local num l_Dia
  local num l_nLegth
  local point l_pBuff
begin
  //矩形

  //根据三个trsf建立frame
  call SetFrame(x_trSource,l_fFrame,x_bRes)
  if !x_bRes
    return
  endIf


  //矩形的宽
  l_Dia=distance(x_trSource[1],x_trSource[2])
  //矩形的长
  l_nLegth=distance(x_trSource[0],x_trSource[1])



  link(l_pBuff,l_fFrame)
  l_pBuff.trsf={l_nLegth/2,0,0,0,0,0}
  x_trDest[0]=position(l_pBuff,world)

  l_pBuff.trsf={l_nLegth,0,0,0,0,0}
  x_trDest[1]=position(l_pBuff,world)

  l_pBuff.trsf={l_nLegth,l_Dia,0,0,0,0}
  x_trDest[2]=position(l_pBuff,world)

  l_pBuff.trsf={0,l_Dia,0,0,0,0}
  x_trDest[3]=position(l_pBuff,world)


  l_pBuff.trsf={0,0,0,0,0,0}
  x_trDest[4]=position(l_pBuff,world)

  x_trDest[5]=x_trDest[0]

    //圆心点
  l_pBuff.trsf={l_nLegth/2,min(l_nLegth/2,l_Dia/2),0,0,0,0}
  x_trDest[20]=position(l_pBuff,world)


end

--- RegulPoint.pgx ---
public program RegulPoint(trsf& x_trSource[], num x_nType, trsf x_trDownLead, point& x_pCut[], point& x_pMc[], bool& x_bMc[], trsf& x_trPara[], bool& x_bRes, bool x_bWeld)
  local num l_nPointCout
  local num l_nNum
  local trsf l_trCutIn[2]
  local trsf l_trCutOut[2]
  local trsf l_trPara[3]
  local num l_nBuff
  local trsf l_trSupport
  local trsf l_trBuff[2]
  local trsf l_trWeld[3]
begin
  //规则图形运动点算法
  //图形类型
  //根据示教的点数来确定运行的点数
  //trCut[20]作为规则图形的中心点
  //如果添加新的类型，只需在Algorith中添加，只支持三个点建立标准图形

  //参数初始化与参数合法化判断
  //x_type 图形类型

  //除了切圆管外，其他图形所有的姿态RX,RY,RZ,都是一样的，可以称为平面图形

  //三点法第一点是切入点
  //第二点是切割点
  //第三点是圆弧的参数


  //2015.02.12
  //添加新的路径
  if x_nType==9
    x_bRes=true
    return
  endIf




  //参数初始化
  x_bRes=false
  resize(trCut,1,100)

  //判断传入参数合法性
  if x_trDownLead.x<0 or x_trDownLead.x>3 or x_trDownLead.z<0 or x_trDownLead.z>3
    return
  endIf

  //保留最初的运动参数
  for l_nNum=0 to min(size(x_trPara)-1,2)
    l_trPara[l_nNum]=x_trPara[l_nNum]
  endFor

  //强制取消切入与切出]
  if x_bWeld
    x_trDownLead.x=x_trDownLead.z=0
  endIf



  //用来获得规则图形转换为movel movec的点数
  switch x_nType

    //圆 三点法
    case 1,11
      l_nPointCout=3
      call Circumcircle(x_trSource,l_trSupport,l_nNum,x_bRes)
      if !x_bRes

        return
      endIf
      //*******************************
      //2014.4.8
      //为焊接
      if x_bWeld and x_trDownLead.rz!=36 and x_trDownLead.rz>0
        call Cshape(x_trSource,trCut,x_trDownLead.rz*10,l_nPointCout,l_trSupport,l_nNum,x_bRes)

        if !x_bRes
          return
        endIf
        //*******************************
      else
        call CirClePoint(l_trSupport,l_nNum,trCut,x_bRes)
      endIf
    break




    //圆 圆心直径法
    case 2,12
      l_nPointCout=3
      l_trSupport=x_trSource
      call CirClePoint(x_trSource,x_trDownLead.ry,trCut,x_bRes)
      //***********************************
      //2014.4.8
      //为焊接
      if x_bWeld and x_trDownLead.rz!=36 and x_trDownLead.rz>0
        l_trWeld[0]=trCut[0]
        l_trWeld[1]=trCut[1]
        l_trWeld[2]=trCut[2]
        call Cshape(l_trWeld,trCut,x_trDownLead.rz*10,l_nPointCout,l_trSupport,x_trDownLead.ry,x_bRes)
        if !x_bRes
          return
        endIf
      endIf
      //*************************************
    break



    //三角形
    case 3,13
      l_nPointCout=5
      call TrianglePoint(x_trSource,trCut,x_bRes)
    break

    //矩形
    case 4,14
      l_nPointCout=6
      call RectanglePoint(x_trSource,trCut,x_bRes)
    break

    //五边形
    case 5,15
      l_nPointCout=7
      call PentagonPoint(x_trSource,trCut,x_bRes)
    break

    //六边形
    case 6,16
      l_nPointCout=8
      call HexagonPoint(x_trSource,trCut,x_bRes)
    break

    //腰形孔
    case 7,17
      l_nPointCout=6
      call EllipsePoint(x_trSource,trCut,x_bRes)
    break
    //五角星
    case 21
      l_nPointCout=11
      x_trDownLead.x=x_trDownLead.z=0
      call PentaclePoint(x_trSource,trCut,x_bRes)
    break

    // 切圆管
    case 22
      l_nPointCout=3
      x_trDownLead.x=x_trDownLead.z=0
      call TubePoint(x_trSource,x_trDownLead.rz,trCut,x_bRes)
    break


    //C型-三点法
    case 24
      x_trDownLead.x=x_trDownLead.z=0
      call Circumcircle(x_trSource,l_trSupport,l_nNum,x_bRes)
      if !x_bRes
        return
      endIf
      call Cshape(x_trSource,trCut,x_trDownLead.rz*10,l_nPointCout,l_trSupport,l_nNum,x_bRes)
      if !x_bRes
        return
      endIf
    break


    //默认退出，没有定义的图形序号则报错退出
    default
      return
    break

  endSwitch

  //××××××××××××××××××××××××××××××××××××××××××××××××××××××××××××××××××××××××
  //引线处理


  //××××××××××××××××××××××××××××××××××××××××
  //2014.10.23
  //如果引线长度是101，则认为是厚板切割
  //按照厚板切割程序进行
  if x_trDownLead.x!=0 and x_trDownLead.y==101
    x_trDownLead.x=1
  endIf
  //××××××××××××××××××××××××××××××××××××××××××



  //引线点数
  l_nPointCout=l_nPointCout+sel(x_trDownLead.x>0,1,0)+sel(x_trDownLead.z>0,1,0)
  //把原来运动参数保留



  //对数组大小进行重新分配
  resize(x_pCut,1,l_nPointCout)
  resize(x_pMc,1,l_nPointCout)
  resize(x_bMc,1,l_nPointCout)
  resize(x_trPara,1,l_nPointCout)

  l_nPointCout=l_nPointCout-sel(x_trDownLead.x>0,1,0)-sel(x_trDownLead.z>0,1,0)
  //对于点数进行规划


  //根据图形中心点与第一个和第二个点来获得切入切出线点
  l_trBuff[0]=trCut[0]
  l_trBuff[1]=trCut[1]

  switch x_nType
    case  11,12,1,2
      l_trBuff[1]=trCut[9]
    break
  endSwitch

  //默认内切
  //切入点
  //l_tr
  call CutIn(trCut[20],l_trBuff,l_trCutIn,l_trSupport,x_trDownLead.x,x_trDownLead.y,x_bRes)
  if !x_bRes
    return
  endIf

  //切出点
  call CutOut(trCut[20],l_trBuff,l_trCutOut,l_trSupport,x_trDownLead.z,x_trDownLead.rx,x_bRes)
  if !x_bRes
    return
  endIf


  l_trBuff[0]=trCut[0]
  l_trBuff[1]=trCut[1]

  switch x_nType

    case  11,12,1,2
      l_trBuff[1]=trCut[9]
    break
  endSwitch


  //外切图形
  switch  x_nType

    case 11,12,13,14,15,16,17,18

      if x_trDownLead.x>0
        call LineSymArray(l_trCutIn,l_trBuff,l_trCutIn,x_bRes)
        if !x_bRes
          return
        endIf
      endIf

      if x_trDownLead.z>0
        call LineSymArray(l_trCutOut,l_trBuff,l_trCutOut,x_bRes)
        if !x_bRes
          return
        endIf
      endIf
    break

  endSwitch



  //****************************************************
  //******************************************************


  //进行点数的赋值
  //参数初始化
  for l_nNum=0 to size(x_bMc)-1
    x_bMc[l_nNum]=false
    // x_trPara[l_nNum]=l_trPara[0]
  endFor
  //切入
  switch x_trDownLead.x
    //无
    case 0
      x_pCut[0].trsf=trCut[0]

    break
    //直线
    case 1
      x_pCut[0].trsf=l_trCutIn[0]
      x_pCut[1].trsf=trCut[0]
    break

    //圆弧
    case 2
      x_pCut[0].trsf=l_trCutIn[0]
      x_pMc[1].trsf=l_trCutIn[1]
      x_pCut[1].trsf=trCut[0]
      x_bMc[1]=true
    break
  endSwitch

  //切割点
  //主要是有圆弧点的判断
  switch x_nType
    //圆
    case 1,11,2,12,22
      //焊接
      //2014.4.8
      if x_bWeld and x_trDownLead.rz!=36 and x_trDownLead.rz>0
        for l_nNum=1 to l_nPointCout-1
          x_pMc[l_nNum].trsf=trCut[l_nNum*2-1]
          x_pCut[l_nNum].trsf=trCut[l_nNum*2]

          x_bMc[l_nNum]=true
        endFor
      else
        //*************************************************
        x_pMc[sel(x_trDownLead.x>0,1,0)+1].trsf=trCut[1]
        x_pCut[sel(x_trDownLead.x>0,1,0)+1].trsf=trCut[2]
        x_bMc[sel(x_trDownLead.x>0,1,0)+1]=true

        x_pMc[sel(x_trDownLead.x>0,1,0)+2].trsf=trCut[3]
        x_pCut[sel(x_trDownLead.x>0,1,0)+2].trsf=trCut[4]

        x_bMc[sel(x_trDownLead.x>0,1,0)+2]=true

      endIf


    break

    //腰形
    case 7,17

      x_pCut[sel(x_trDownLead.x>0,1,0)+1].trsf=trCut[1]
      x_pMc[sel(x_trDownLead.x>0,1,0)+2].trsf=trCut[2]
      x_pCut[sel(x_trDownLead.x>0,1,0)+2].trsf=trCut[3]
      x_bMc[sel(x_trDownLead.x>0,1,0)+2]=true

      x_pCut[sel(x_trDownLead.x>0,1,0)+3].trsf=trCut[4]
      x_pCut[sel(x_trDownLead.x>0,1,0)+4].trsf=trCut[6]
      x_pMc[sel(x_trDownLead.x>0,1,0)+4].trsf=trCut[5]
      x_bMc[sel(x_trDownLead.x>0,1,0)+4]=true

      x_pCut[sel(x_trDownLead.x>0,1,0)+5].trsf=trCut[7]
    break


    //C形
    case 24
      for l_nNum=1 to l_nPointCout-1
        x_pMc[l_nNum].trsf=trCut[l_nNum*2-1]
        x_pCut[l_nNum].trsf=trCut[l_nNum*2]

        x_bMc[l_nNum]=true
      endFor
    break

    default
      for l_nNum=1 to  l_nPointCout-1
        x_pCut[sel(x_trDownLead.x>0,1,0)+l_nNum].trsf=trCut[l_nNum]
      endFor

    break


  endSwitch



  //切出
  switch x_trDownLead.z
    case 1
      x_pCut[size(x_pCut)-1].trsf=l_trCutOut[0]
    break

    case 2
      x_pCut[size(x_pCut)-1].trsf=l_trCutOut[0]
      x_pMc[size(x_pCut)-1].trsf=l_trCutOut[1]
      x_bMc[size(x_pCut)-1]=true
    break
  endSwitch



  //××××××××××××××××××××××××××××××××
  //三点建立顺时针或者逆时针时的姿态
  //  call GetClockwise(x_trSource,l_trBuff,x_bRes)
  //
  //  if x_nType!=22 and x_nType!=11 and x_nType!=1  and x_bRes
  //    for l_nNum=0 to size(x_pCut)-1
  //      x_pMc[l_nNum].trsf.rx=x_pCut[l_nNum].trsf.rx=l_trBuff[0].rx
  //      x_pMc[l_nNum].trsf.ry=x_pCut[l_nNum].trsf.ry=l_trBuff[0].ry
  //      x_pMc[l_nNum].trsf.rz=x_pCut[l_nNum].trsf.rz=l_trBuff[0].rz
  //
  //    endFor


  //endIf

  //*********************************************************


  //切割参数的分配
  //类型2 只有一个点
  x_trPara[0]=l_trPara[0]
  for l_nBuff=1 to size(x_trPara)-1
    x_trPara[l_nBuff]=l_trPara[sel(x_nType==2 or x_nType==12,0,1)]
  endFor

  //2014.6.23  把第一点的参数强制赋值给切入点
  if x_trDownLead.x==1 or x_trDownLead.x==2
    x_trPara[1]=l_trPara[0]
  endIf




  //腰形孔
  //把圆弧段的参数利用第三点的参数
  if x_nType==7 or x_nType==17
    for l_nBuff=0 to size(x_pCut)-1
      if x_pCut[l_nBuff].trsf==trCut[1] or x_pCut[l_nBuff].trsf==trCut[3]
        x_trPara[l_nBuff]=l_trPara[2]
      endIf
    endFor
  endIf



  //强制所有规则图形的姿态
  for l_nBuff=0 to size(x_pCut)-1
    x_pMc[l_nBuff].trsf.rx=x_pCut[l_nBuff].trsf.rx=x_trSource.rx
    x_pMc[l_nBuff].trsf.ry=x_pCut[l_nBuff].trsf.ry=x_trSource.ry
    x_pMc[l_nBuff].trsf.rz= x_pCut[l_nBuff].trsf.rz=x_trSource.rz

  endFor


  x_bRes=true
end

--- SETFRAME.pgx ---
public program SetFrame(trsf& x_trSource[], frame& x_fFrame, bool& x_bRes)
  local point l_pPoint[3]
  local num l_ni
  local bool l_bIn
begin
  //把三个trsf转换为frame
  //如果x_frame是局部变量,需要在建立的程序中先link
  link(x_fFrame,world)
  x_fFrame.trsf={0,0,0,0,0,0}
  x_bRes=false
  if size(x_trSource)<3
    return
  endIf


  //建立frame
  for l_ni=0 to 2
    l_pPoint[l_ni].trsf=x_trSource[l_ni]
    link(l_pPoint[l_ni],world)
  endFor

  x_bRes=setFrame(l_pPoint[0],l_pPoint[1],l_pPoint[2],x_fFrame)==0


end

--- TrianglePoint.pgx ---
public program TrianglePoint(trsf& x_trSource[], trsf& x_trDest[], bool& x_bRes)
  local frame l_fFrame
  local trsf l_trCenter
  local num l_nDia
  local point l_p
  local trsf l_trBuff[3]
begin
  //三角形三点
  call Inscribedcircle(x_trSource,l_trCenter,l_nDia,x_bRes)
  if !x_bRes
    return
  endIf
      //圆心点
  x_trDest[20]=l_trCenter

  call SetFrame(x_trSource,l_fFrame,x_bRes)
  if !x_bRes
    return
  endIf

  l_p.trsf=l_trCenter
  link(l_p,world)
  l_p.trsf=position(l_p,l_fFrame)
  l_p.trsf.y=0
  link(l_p,l_fFrame)
  x_trDest[0]=position(l_p,world)

  x_trDest[1]=x_trSource[1]
  x_trDest[2]=x_trSource[2]
  x_trDest[3]=x_trSource[0]
  x_trDest[4]=x_trDest[0]

  for l_nDia=0 to 4
    x_trDest[l_nDia].rx= x_trDest[0].rx
    x_trDest[l_nDia].ry = x_trDest[0].ry
    x_trDest[l_nDia].rz= x_trDest[0].rz
  endFor



end

--- TubePoint.pgx ---
public program TubePoint(trsf& x_trSource[], num x_nAngle, trsf& x_trDest[], bool& x_bRes)
  local num l_ni
  local frame l_fFrame
  local num l_Dia
  local point l_pBuff
  local trsf l_trSupport
  local trsf l_trBuff[3]
begin
 //切管子应用
 //设置三点和一个角度就可以进行实现

  call Circumcircle(x_trSource,l_trSupport,l_Dia,x_bRes)
  if !x_bRes
    return
  endIf
  call CirClePoint(l_trSupport,l_Dia,x_trDest,x_bRes)
  if !x_bRes
    return
  endIf
  x_trDest[20]=l_trSupport




  //对点在对应坐标系下进行偏移
  for l_ni=0 to 3
    l_trBuff[0]=x_trDest[l_ni]
    l_trBuff[1]=l_trSupport
    l_trBuff[2]=x_trDest[l_ni+1]
    call SetFrame(l_trBuff,l_fFrame,x_bRes)
    if !x_bRes
      return
    endIf
    l_pBuff.trsf=x_trDest[l_ni]
    link(l_pBuff,world)
   l_pBuff=compose(l_pBuff,l_fFrame,{0,0,0,0,-x_nAngle,0})
    x_trDest[l_ni]=position(l_pBuff,world)
  endFor
  x_trDest[4]=x_trDest[0]


end
